// TwinCAT 3 PLC project Robotino_PLC
// ProgramVersion: 3.1.4022.0
// libraries:
//   Tc2_EtherCAT, * (Beckhoff Automation GmbH)
//   Tc2_SerialCom, * (Beckhoff Automation GmbH)
//   Tc2_Standard, * (Beckhoff Automation GmbH)
//   Tc2_System, * (Beckhoff Automation GmbH)
//   Tc2_Utilities, * (Beckhoff Automation GmbH)
//   Tc3_Module, * (Beckhoff Automation GmbH)
// project tree:
//   DUTs/ EnumState.TcDUT
//   / PlcTask.TcTTO
//   POUs/COE_Auswertung/ PDODatenMotor.TcPOU, SDODatenMotor.TcPOU, getSDODatenMotor.TcPOU, getSDOMotorErrorFlags.TcPOU, getSDODatenMotorklemme.TcPOU, SDOMotorErrorFlags.TcPOU
//   POUs/Greiferansteuerung/ Greiferansteuerung.TcPOU
//   POUs/Motoransteuerung/ Motoransteuerung.TcPOU
//   POUs/Motormesswerte/ Motormesswerte.TcPOU
//   POUs/RS232/ BackgroundPcCOM.TcPOU, FB_SerialCom.TcPOU, RS232_Communication.TcPOU
//   POUs/Shutdown/ Shutdown.TcPOU
//   POUs/UDP/ UDP.TcPOU, UDPConnect.TcPOU
// real-time tasks:
//   TASK IrSensorTask: cycle T#1ms, priority 2, ADS port 351
//   TASK UdpTask: cycle T#2ms, priority 3, ADS port 355
//   TASK SimulinkTask: cycle T#5ms, priority 4, ADS port 353
//   TASK PlcTask1: cycle T#400us, priority 1, ADS port 352
// I/O:
//   DEVICE Robotino SPS, AmsNetId 192.168.0.109.2.1
//     Klemme 1 (EK1200) [EK1200-5000 EtherCAT Netzteil (2A E-Bus)]
//       Motorklemme 1 [EL7342 2K. DC-Motor-Endstufe (50V, 3.5A)]
//       Motorklemme 2 [EL7342 2K. DC-Motor-Endstufe (50V, 3.5A)]
//       Digitale Eingänge [EL1008 8K. Dig. Eingang 24V, 3ms]
//       Digitale Ausgänge [EL2004 4K. Dig. Ausgang 24V, 0.5A]
//       Analoge Eingänge (8) [EL3068 8K. Ana. Eingang 0-10V]
//       Analog Eingänge (4) [EL3064 4K.Ana. Eingang 0-10V]
//       Netzklemme (5V) [EL9505 Netzteilklemme 5V]
//       Busendklemme [EL9011 Endklemme]
//   DEVICE UDP Adapter
//   DEVICE RS232
// variable links:
//   Robotino SPS <-> TcCOM Objects/Object2 (Gewerk3_Simulink_Regler)
//     Term 1 (EK1200)/Digitale Eingänge/Channel 2/Bumper <-> Input/processData[14]
//   Robotino SPS <-> irSensors/irSensors_Obj
//     Term 1 (EK1200)/Analog Eingänge (4)/AI Standard Channel 1/IR9 <-> Inputs/irInputData[8]
//     Term 1 (EK1200)/Analoge Eingänge (8)/AI Standard Channel {1..8}/IR{1..8} <-> Inputs/irInputData[{0..7}]  (8 links)
//   Robotino_PLC/Robotino_PLC Instance <-> RS232
//     PlcTask Inputs/BackgroundPcCOM.stIn_PcCom/D[{0..63}] <-> Inputs/Data{1..64}  (64 links)
//     PlcTask Inputs/BackgroundPcCOM.stIn_PcCom/SerStatus <-> Inputs/Status
//     PlcTask Outputs/BackgroundPcCOM.stOut_PcCom/D[{0..63}] <-> Outputs/Data{1..64}  (64 links)
//     PlcTask Outputs/BackgroundPcCOM.stOut_PcCom/SerCtrl <-> Outputs/Ctrl
//   Robotino_PLC/Robotino_PLC Instance <-> Robotino SPS/Term 1 (EK1200)/Analog Eingänge (4)
//     PlcTask Inputs/Shutdown.cell1 <-> AI Standard Channel 2/Zelle1
//     PlcTask Inputs/Shutdown.cell12 <-> AI Standard Channel 3/Zelle12
//   Robotino_PLC/Robotino_PLC Instance <-> Robotino SPS/Term 1 (EK1200)/Digitale Eingänge
//     PlcTask Inputs/Greiferansteuerung.greiferLichtschrankeFromIO <-> Channel 6/Lichtschranke
//     PlcTask Inputs/Greiferansteuerung.greiferSliderFromIO <-> Channel 5/Greifer
//     PlcTask Inputs/Motoransteuerung.bumper <-> Channel 2/Bumper
//     PlcTask Inputs/Shutdown.shutdownButton <-> Channel 8/Shutdown
//   Robotino_PLC/Robotino_PLC Instance <-> Robotino SPS/Term 1 (EK1200)/Motorklemme 1
//     PlcTask Inputs/Motormesswerte.encDataFromMotor1 <-> ENC Status compact Channel 1/Counter value
//     PlcTask Inputs/Motormesswerte.encDataFromMotor2 <-> ENC Status compact Channel 2/Counter value
//     PlcTask Inputs/PDODatenMotor.SpannungPDOMotor1 <-> DCM Synchron info data Channel 1/SpannungM1
//     PlcTask Inputs/PDODatenMotor.SpannungPDOMotor2 <-> DCM Synchron info data Channel 2/SpannungM2
//     PlcTask Inputs/PDODatenMotor.StromPDOMotor1 <-> DCM Synchron info data Channel 1/StromM1
//     PlcTask Outputs/Motoransteuerung.enableToMotor1 <-> DCM Control Channel 1/Control/Enable
//     PlcTask Outputs/Motoransteuerung.enableToMotor2 <-> DCM Control Channel 2/Control/Enable
//     PlcTask Outputs/Motoransteuerung.velocityToMotor1 <-> DCM Velocity Channel 1/Velocity
//     PlcTask Outputs/Motoransteuerung.velocityToMotor2 <-> DCM Velocity Channel 2/Velocity
//   Robotino_PLC/Robotino_PLC Instance <-> Robotino SPS/Term 1 (EK1200)/Motorklemme 2
//     PlcTask Inputs/Motormesswerte.encDataFromMotor3 <-> ENC Status compact Channel 1/Counter value
//     PlcTask Inputs/PDODatenMotor.SpannungPDOGreifer <-> DCM Synchron info data Channel 2/SpannungGreifer
//     PlcTask Inputs/PDODatenMotor.SpannungPDOMotor3 <-> DCM Synchron info data Channel 1/SpannungM3
//     PlcTask Inputs/PDODatenMotor.StromPDOGreifer <-> DCM Synchron info data Channel 2/StromGreifer
//     PlcTask Outputs/Greiferansteuerung.greiferEnable <-> DCM Control Channel 2/Control/Enable
//     PlcTask Outputs/Greiferansteuerung.greiferValue <-> DCM Velocity Channel 2/Velocity
//     PlcTask Outputs/Motoransteuerung.enableToMotor3 <-> DCM Control Channel 1/Control/Enable
//     PlcTask Outputs/Motoransteuerung.velocityToMotor3 <-> DCM Velocity Channel 1/Velocity
//   Robotino_PLC/Robotino_PLC Instance <-> TcCOM Objects/Object2 (Gewerk3_Simulink_Regler)
//     PlcTask Inputs/Greiferansteuerung.greiferSignal <-> Output/Grabber
//     PlcTask Inputs/Motoransteuerung.vThetaCartesianToMotors <-> Output/vThetaToMotors
//     PlcTask Inputs/Motoransteuerung.vXCartesianToMotors <-> Output/vXToMotors
//     PlcTask Inputs/Motoransteuerung.vYCartesianToMotors <-> Output/vYToMotors
//     PlcTask Outputs/Greiferansteuerung.greiferLichtschrankeToSimulink <-> Input/processData[0]
//     PlcTask Outputs/Greiferansteuerung.greiferSliderToSimulink <-> Input/processData[1]
//     PlcTask Outputs/Motormesswerte.vXCartesianFromMotors <-> Input/processData[2]
//     PlcTask Outputs/Motormesswerte.vYCartesianFromMotors <-> Input/processData[3]
//     PlcTask Outputs/Motormesswerte.vthetaCartesianFromMotors <-> Input/processData[4]
//     PlcTask Outputs/UDP.theta[4] <-> Input/UDP[11]
//     PlcTask Outputs/UDP.x[4] <-> Input/UDP[9]
//     PlcTask Outputs/UDP.y[4] <-> Input/UDP[10]
//   TcCOM Objects/Object2 (Gewerk3_Simulink_Regler) <-> irSensors/irSensors_Obj
//     Input/processData[{5..13}] <-> Outputs/irDistance[{0..8}]  (9 links)

CONFIGURATION Robotino_PLC
    RESOURCE PLC ON TwinCAT3
        TASK PlcTask(INTERVAL := T#400us, PRIORITY := 1);
        PROGRAM SDODatenMotor WITH PlcTask : SDODatenMotor;
        PROGRAM Motormesswerte WITH PlcTask : Motormesswerte;
        PROGRAM UDP WITH PlcTask : UDP;
        PROGRAM Greiferansteuerung WITH PlcTask : Greiferansteuerung;
        PROGRAM Motoransteuerung WITH PlcTask : Motoransteuerung;
        PROGRAM Shutdown WITH PlcTask : Shutdown;
        PROGRAM PDODatenMotor WITH PlcTask : PDODatenMotor;
        PROGRAM RS232_Communication WITH PlcTask : RS232_Communication;
    END_RESOURCE
END_CONFIGURATION

// ---- DUTs/EnumState.TcDUT
{attribute 'qualified_only'}
{attribute 'strict'}
TYPE EnumState :
(
	init,
	drive,
	reset
);
END_TYPE

// ---- POUs/COE_Auswertung/SDODatenMotor.TcPOU
PROGRAM SDODatenMotor
VAR
	DatenMotor1: getSDODatenMotor;
	DatenMotor2: getSDODatenMotor;
	DatenMotor3: getSDODatenMotor;
	
	StromMotor1 AT%Q* : INT;
	StromMotor2 AT%Q* : INT;
	StromMotor3 AT%Q* : INT;
	
	SpannungMotor1 AT%Q*:UINT;
	SpannungMotor2 AT%Q*:UINT;
	SpannungMotor3 AT%Q*:UINT;
	
END_VAR

(*** Daten azyklisch aus Klemme auslesen per SDO
	getSDO* liest CoE-Daten aus der Klemme aus:
		- getSDODatenMotor: Alle Daten, die in Objekt 9020 bzw. 9030 der Motorklemme liegen (siehe Reiter CoE-Daten auf Klemme)
			- Strom/Spannung werden alle 0.4 ms ausgelesen, Rest alle 1 ms
		- getSDODatenMotorklemme: evtl. interessante Klemmendaten, Abruf alle 5 ms
		- getSDOMotorErrorFlags: Fehlerflags wie Kurzschluss, zu hohe Temp, Überlast usw., Abruf alle 5 ms
*)

DatenMotor1.nSlaveAddr := 1001;		// Klemme  1
DatenMotor1.nIndex := 16#9020;		// Channel 1
DatenMotor1();


DatenMotor2.nSlaveAddr := 1001;		// Klemme  1
DatenMotor2.nIndex := 16#9030;		// Channel 2
DatenMotor2();

DatenMotor3.nSlaveAddr := 1002; 	// Klemme  2
DatenMotor3.nIndex := 16#9020;		// Channel 1
DatenMotor3();


StromMotor1 := DatenMotor1.Strom;
StromMotor2 := DatenMotor2.Strom;
StromMotor3 := DatenMotor3.Strom;

SpannungMotor1 :=DatenMotor1.Spannung;
SpannungMotor2 :=DatenMotor2.Spannung;
SpannungMotor3 :=DatenMotor3.Spannung;

END_PROGRAM

// ---- POUs/COE_Auswertung/getSDODatenMotor.TcPOU
FUNCTION_BLOCK getSDODatenMotor
VAR_INPUT
	nSlaveAddr: UINT;
	nIndex: WORD;
END_VAR

VAR_OUTPUT
	// Ausglesene SDOs aus 9020 bzw. 9030
	Spannung: UINT;
	Strom: INT;
	Strombegrenzung: UINT;
	Regelfehler: INT;
	Geschwindigkeit: INT;
	Overloadtime: UINT;
	Overtemperature: BOOL;
	Torqueoverload: BOOL;
	Shortcircuit: BOOL;
END_VAR
	
VAR
	MotorspannungBlock: FB_EcCoESdoRead;	
	MotorstromBlock: FB_EcCoESdoRead;
	StrombegrenzungBlock: FB_EcCoESdoRead;
	RegelfehlerBlock: FB_EcCoESdoRead;
	GeschwindigkeitBlock: FB_EcCoESdoRead;
	OverloadTimeBlock: FB_EcCoESdoRead;
	Short_CircuitBlock: FB_EcCoESdoRead;
	Torque_OverloadBlock: FB_EcCoESdoRead;
	Over_TemperatureBlock: FB_EcCoESdoRead;

	trigger: BOOL;
	triggerStromSpannung: BOOL;
	TON_0: TON;
	TON_1: TON;
	TON_2: TON;
	TON_3: TON;
	ms: TIME;

END_VAR

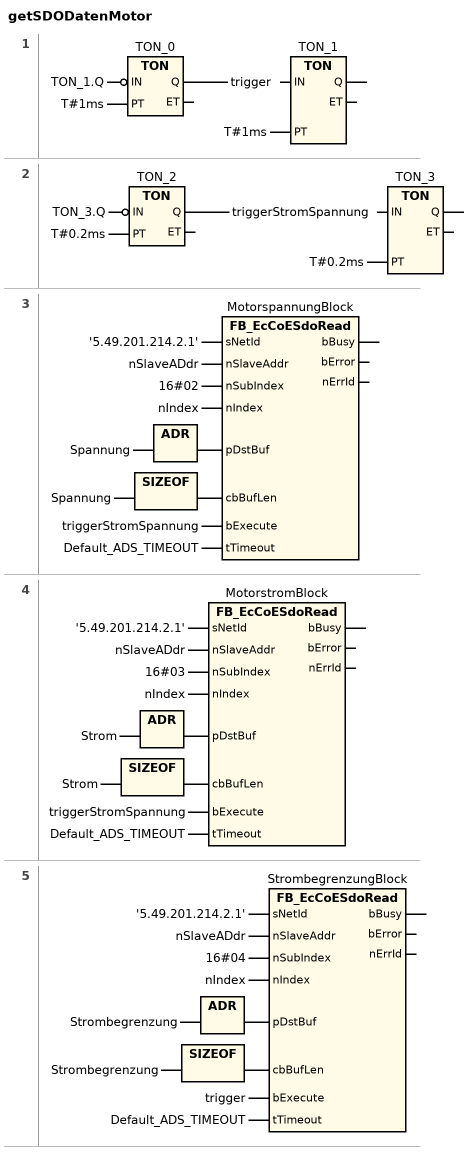
// NETWORK 1
TON_0(IN := NOT TON_1.Q, PT := T#1ms); // TON
trigger := TON_0.Q;
TON_1(IN := TON_0.Q, PT := T#1ms); // TON

// NETWORK 2
TON_2(IN := NOT TON_3.Q, PT := T#0.2ms); // TON
triggerStromSpannung := TON_2.Q;
TON_3(IN := TON_2.Q, PT := T#0.2ms); // TON

// NETWORK 3
MotorspannungBlock(
    sNetId := '5.49.201.214.2.1',
    nSlaveAddr := nSlaveADdr,
    nSubIndex := 16#02,
    nIndex := nIndex,
    pDstBuf := ADR(Spannung),
    cbBufLen := SIZEOF(Spannung),
    bExecute := triggerStromSpannung,
    tTimeout := Default_ADS_TIMEOUT); // FB_EcCoESdoRead

// NETWORK 4
MotorstromBlock(
    sNetId := '5.49.201.214.2.1',
    nSlaveAddr := nSlaveADdr,
    nSubIndex := 16#03,
    nIndex := nIndex,
    pDstBuf := ADR(Strom),
    cbBufLen := SIZEOF(Strom),
    bExecute := triggerStromSpannung,
    tTimeout := Default_ADS_TIMEOUT); // FB_EcCoESdoRead

// NETWORK 5
StrombegrenzungBlock(
    sNetId := '5.49.201.214.2.1',
    nSlaveAddr := nSlaveADdr,
    nSubIndex := 16#04,
    nIndex := nIndex,
    pDstBuf := ADR(Strombegrenzung),
    cbBufLen := SIZEOF(Strombegrenzung),
    bExecute := trigger,
    tTimeout := Default_ADS_TIMEOUT); // FB_EcCoESdoRead

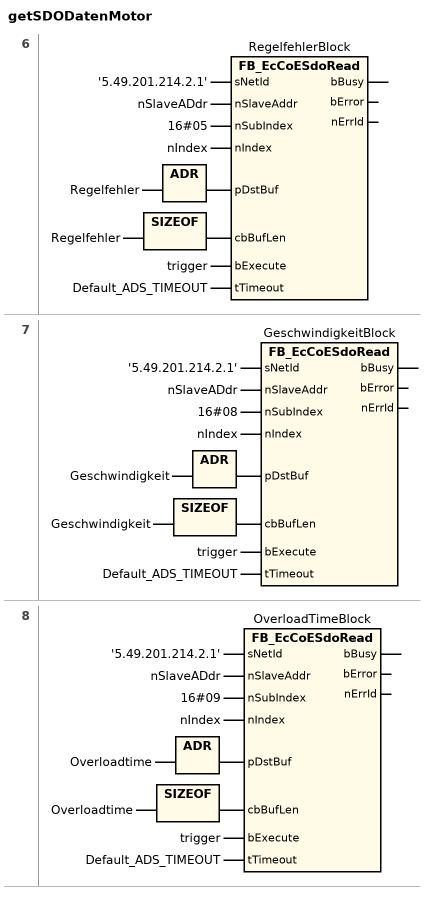
// NETWORK 6
RegelfehlerBlock(
    sNetId := '5.49.201.214.2.1',
    nSlaveAddr := nSlaveADdr,
    nSubIndex := 16#05,
    nIndex := nIndex,
    pDstBuf := ADR(Regelfehler),
    cbBufLen := SIZEOF(Regelfehler),
    bExecute := trigger,
    tTimeout := Default_ADS_TIMEOUT); // FB_EcCoESdoRead

// NETWORK 7
GeschwindigkeitBlock(
    sNetId := '5.49.201.214.2.1',
    nSlaveAddr := nSlaveADdr,
    nSubIndex := 16#08,
    nIndex := nIndex,
    pDstBuf := ADR(Geschwindigkeit),
    cbBufLen := SIZEOF(Geschwindigkeit),
    bExecute := trigger,
    tTimeout := Default_ADS_TIMEOUT); // FB_EcCoESdoRead

// NETWORK 8
OverloadTimeBlock(
    sNetId := '5.49.201.214.2.1',
    nSlaveAddr := nSlaveADdr,
    nSubIndex := 16#09,
    nIndex := nIndex,
    pDstBuf := ADR(Overloadtime),
    cbBufLen := SIZEOF(Overloadtime),
    bExecute := trigger,
    tTimeout := Default_ADS_TIMEOUT); // FB_EcCoESdoRead

END_FUNCTION_BLOCK

// ---- POUs/Motormesswerte/Motormesswerte.TcPOU
PROGRAM Motormesswerte
VAR
bStart: BOOL := FALSE;	
zaehler : UINT := 0;

//ENC Daten Differenzieren für Geschwindigkeit
diffConst:LREAL:=0.0004;//SECONDS
encDataOldMotor1:UINT:=0;
encDataOldMotor2:UINT:=0;
encDataOldMotor3:UINT:=0;

//Koordinatentransformation Weg
skalEnc:LREAL:=0.00766990393;
x1:LREAL:=0;
x2:LREAL:=0;
x3:LREAL:=0;

xFromMotor1:LREAL:=0;
xFromMotor2:LREAL:=0;
xFromMotor3:LREAL:=0;

//Koordinatentransformation Geschwindigkeit
v1:LREAL:=0;
v2:LREAL:=0;
v3:LREAL:=0;
velocityFromMotor1:LREAL:=0;
velocityFromMotor2:LREAL:=0;
velocityFromMotor3:LREAL:=0;

//INPUTS
encDataFromMotor1 AT%I*  :UINT:=0;
encDataFromMotor2 AT%I*  :UINT:=0;
encDataFromMotor3 AT%I*  :UINT:=0;

diff:  INT :=0;
diff1: INT := 0;
diff2: INT := 0;
diff3: INT := 0;

//OUTPUTS
posXCartesianFromMotors AT%Q*:LREAL:=0;
posYCartesianFromMotors AT%Q*:LREAL:=0;
posThetaCartesianFromMotors AT%Q*:LREAL:=0;

vXCartesianFromMotors AT%Q*:LREAL:=0;
vYCartesianFromMotors AT%Q*:LREAL:=0;
vthetaCartesianFromMotors AT%Q*:LREAL:=0;
END_VAR

IF bStart = FALSE THEN
	encDataOldMotor1 := encDataFromMotor1;
	encDataOldMotor2 := encDataFromMotor2;
	encDataOldMotor3 := encDataFromMotor3;
	bStart := TRUE;
END_IF



// Encoder Wegberechnung und Differenzierung für Geschwindigkeit
diff1:=UINT_TO_INT(encDataFromMotor1) - UINT_TO_INT(encDataOldMotor1);
IF diff1 >= 32767 OR diff1 <= -32767 THEN
	diff1 := 0;
	zaehler := zaehler + 1;
END_IF
diff2:=UINT_TO_INT(encDataFromMotor2) - UINT_TO_INT(encDataOldMotor2);
IF diff2 >= 32767 OR diff2 <= -32767 THEN
	diff2 := 0;
END_IF
diff3:=UINT_TO_INT(encDataFromMotor3) - UINT_TO_INT(encDataOldMotor3);
IF diff3 >= 32767 OR diff3 <= -32767 THEN
	diff3 := 0;
END_IF

xFromMotor1:=xFromMotor1+diff1*skalEnc;
velocityFromMotor1:=diff1/diffConst*skalEnc;

xFromMotor2:=xFromMotor2+diff2*skalEnc;
velocityFromMotor2:=diff2/diffConst*skalEnc;

xFromMotor3:=xFromMotor3+diff3*skalEnc;
velocityFromMotor3:=diff3/diffConst*skalEnc;

// Koordinatentransformation Weg
x1:=-xFromMotor1;
x2:=-xFromMotor2;
x3:=-xFromMotor3;

posXCartesianFromMotors:=(x3 - x1) / (2.0 * COS(30.0*PI/180));  //in mm / s
posYCartesianFromMotors:=(x1 - 2.0 * x2 + x3) / 3.0;            //in mm / s
posThetaCartesianFromMotors:=(x1 + x2 + x3) / (3.0 * 135.0);    //in rad / s

// Koordinatentransformation Geschwindigkeit
v1:=-velocityFromMotor1;
v2:=-velocityFromMotor2;
v3:=-velocityFromMotor3;

vXCartesianFromMotors:=(v3 - v1) / (2.0 * COS(30.0*PI/180));  //in mm / s
vYCartesianFromMotors:=(v1 - 2.0 * v2 + v3) / 3.0;            //in mm / s
vThetaCartesianFromMotors:=(v1 + v2 + v3) / (3.0 * 135.0);    //in rad / s

// Alte Encoderdaten speichern

encDataOldMotor1:=encDataFromMotor1;
encDataOldMotor2:=encDataFromMotor2;
encDataOldMotor3:=encDataFromMotor3;

END_PROGRAM

// ---- POUs/UDP/UDP.TcPOU
PROGRAM UDP

VAR_INPUT
	x	  AT%Q*	: ARRAY[1..4] OF LREAL;
	y	  AT%Q*	: ARRAY[1..4] OF LREAL;
	theta AT%Q*	: ARRAY[1..4] OF LREAL;
END_VAR

VAR
	udp1 : UDPConnect;
	count :INT :=0;
END_VAR

(*** UDP Kommunikation ***
	Hier wird nur der FB UDPConnect instanziert
	Für x,y,theta reichen eigentlich 8 Byte Variablen. Hier: LREAL wegen Kompatibilität
		zu Simulink Regler, der double (=LREAL) als Input braucht
*)

udp1();

END_PROGRAM

// ---- POUs/UDP/UDPConnect.TcPOU
{attribute 'c++_compatible'}
FUNCTION_BLOCK UDPConnect IMPLEMENTS ITcIoUdpProtocolRecv
VAR_INPUT
END_VAR
VAR_OUTPUT
END_VAR

VAR
	{attribute 'TcInitSymbol'}
    oid:              OTCID; 
    ipUdp:            ITcIoUdpProtocol;
    updPort:          UINT := 25000;
    nReceivedPakets:  UINT;
    hrInit :          HRESULT;
    hrSend :          HRESULT;
	
	
END_VAR

// CheckReceived() ruft ReceiveData auf

IF ipUdp <> 0 THEN
    ipUdp.CheckReceived();
END_IF

METHOD FB_exit : BOOL
VAR_INPUT
	bInCopyCode : BOOL; // if TRUE, the exit method is called for exiting an instance that is copied afterwards (online change).
END_VAR
// Destruktor für UDPConnect

IF (NOT bInCopyCode AND ipUdp <> 0) THEN //Shutdown
     ipUdp.UnregisterReceiver(updPort);
    FW_SafeRelease(ADR(ipUdp));
     FB_exit := TRUE;
ELSE
     FB_exit := FALSE;
END_IF
END_METHOD

METHOD FB_init : BOOL
VAR_INPUT
	bInitRetains : BOOL; // if TRUE, the retain variables are initialized (warm start / cold start)
	bInCopyCode : BOOL;  // if TRUE, the instance afterwards gets moved into the copy code (online change)
END_VAR

VAR
    ipSrv: ITComObjectServer;
    hr : HRESULT;
END_VAR
// Konstruktor für UDPConnect

IF NOT bInCopyCode THEN // no online change
    IF ipUdp = 0 THEN
     hrInit := FW_ObjMgr_GetObjectInstance(   oid:=oid, 
    
    iid:=TC_GLOBAL_IID_LIST.IID_ITcIoUdpProtocol, 

    pipUnk:=ADR(ipUdp) );
        IF ( SUCCEEDED(hr) AND ipUdp.RegisterReceiver(updPort, THIS^) = 0 ) THEN //open port
            FB_init := TRUE;
        ELSE
            FB_init := FALSE; 
            FW_SafeRelease(ADR(ipUdp));
        END_IF
    END_IF
END_IF
END_METHOD

METHOD FB_reinit : BOOL
VAR_INPUT
END_VAR
IF (ipUdp <> 0) THEN 
 ipUdp.RegisterReceiver(updPort, THIS^);
END_IF
END_METHOD

{attribute 'object_name' := 'ReceiveData'}
{attribute 'c++_compatible'}
{attribute 'signature_flag' := '33554688'}
{attribute 'pack_mode' := '4'}
{attribute 'show'}
{attribute 'minimal_input_size' := '4'}
METHOD ReceiveData : HRESULT
VAR_INPUT
	ipAddr	: UDINT;
	udpDestPort	: UINT;
	udpSrcPort	: UINT;
	nData	: UDINT;
	pData	: PVOID;	// Pointer auf Datenbereich des UDP-Pakets
	pVlan	: POINTER TO ETYPE_VLAN_HEADER := 0;
END_VAR

VAR
	i	: ULINT := 0;
END_VAR
nReceivedPakets := nReceivedPakets+1; 	// zählt Pakete

(*** Auslesen des Datenbereichs von UDP-Paketen ***
	* UDP-Telegramm besteht aus 56*8 = 448 Bytes (siehe UDP-Doku Lokalisierungsrechner)
	  Pro Robotino: 3*8 = 24 Bytes: je 8 Bytes für x-Koord, y-Koord, theta in rad
	  Robotino1: Bytes 1-8   -> x-Koord, Bytes 9-16  -> y-Koord, Bytes 17-24 -> theta
	  Robotino2: Bytes 25-32 -> x-Koord, Bytes 33-40 -> y-Koord, Bytes 41-48 -> theta  usw.. 
	* pData zeigt auf Adressbereich, in dem die 448 Byte großen UDP-Daten liegen
	  in der Schleife werden jeweils 8 Byte in den UDP-Array geschrieben und der Pointer nach
	  jedem Schritt um 8 Byte weiter geschoben
*)

// 4 Schleifendurchgänge für 4 Robotinos, i=0 -> Robo1 i=1 -> Robo2 usw..
FOR i := 0 TO 3 DO
	memcpy(ADR(UDP.x[i+1]),pData+((i*3)*8),8);			// x-Koord
	memcpy(ADR(UDP.y[i+1]),pData+((i*3+1)*8),8);		// y-Koord
	memcpy(ADR(UDP.theta[i+1]),pData+((i*3+2)*8),8);	// theta
END_FOR;
END_METHOD

{attribute 'c++_compatible'}
{attribute 'minimal_input_size' := '4'}
{attribute 'pack_mode' := '4'}
{warning 'Methodenimplementierung hinzufügen'}
METHOD TcAddRef : UDINT
END_METHOD

{attribute 'c++_compatible'}
{attribute 'minimal_input_size' := '4'}
{attribute 'pack_mode' := '4'}
{warning 'Methodenimplementierung hinzufügen'}
METHOD TcQueryInterface : HRESULT
VAR_INPUT
	iid	: REFERENCE TO IID;
	pipItf	: POINTER TO PVOID;
END_VAR
END_METHOD

{attribute 'c++_compatible'}
{attribute 'minimal_input_size' := '4'}
{attribute 'pack_mode' := '4'}
{warning 'Methodenimplementierung hinzufügen'}
METHOD TcRelease : UDINT
END_METHOD

END_FUNCTION_BLOCK

// ---- POUs/Greiferansteuerung/Greiferansteuerung.TcPOU
PROGRAM Greiferansteuerung
VAR
	greiferSignal AT%I*:LREAL:=0;
	greiferEnable AT%Q*:BOOL:=0;
	greiferValue  AT%Q* :INT:=0;
	
	greiferSliderFromIO 	AT%I*:BOOL:=0;
	greiferSliderToSimulink AT%Q*:LREAL:=0;
	
	greiferLichtschrankeFromIO AT%I*:BOOL:=0;
	greiferLichtschrankeToSimulink AT%Q*:LREAL:=0;
END_VAR

IF greiferSignal=0 THEN
	greiferEnable:=1;
	greiferValue:=-32767;
ELSE
	greiferEnable:=1;
	greiferValue:=32767;
END_IF

greiferSliderToSimulink:=BOOL_TO_LREAL(NOT(greiferSliderFromIO));
greiferLichtschrankeToSimulink:=BOOL_TO_LREAL(NOT(greiferLichtschrankeFromIO));

END_PROGRAM

// ---- POUs/Motoransteuerung/Motoransteuerung.TcPOU
PROGRAM Motoransteuerung
VAR	
	//Zustandsautomat
	state:		EnumState:=EnumState.init;
	nextState:	EnumState:=EnumState.init;

	//Achsen Freischalten
	
	enableMotors: BOOL	:=0;

	//Umgerechnete Werte
	vX:		LREAL:=0;
	vY:		LREAL:=0;
	vTheta:	LREAL:=0;

	//Fahrrichtung Motor
	velocityMotor1 :LREAL:=0;
	velocityMotor2 :LREAL:=0;
	velocityMotor3 :LREAL:=0;
	
	//Skalierung auf MaxGeschwindigkeit Skalierung hängt mit CoE Register 8020:07 8020:08 zusammen !!!
	velocityMax:LREAL:=942.4777961;// Nenndrehzahl U/min CoE Register 8020:07 8020:08 fesgelegt Faktor 16 Wegen Getriebe 1:16
	velocityMotorsTf:LREAL:=0;
	
	// Skalierung auf Ansteuersignale LREAL=>WORD   Skalierung hängt mit CoE Register 8020:07 8020:08 zusammen !!!
	skalPos:LREAL:=34.7668668;//  MaxValue/MaxVelocity   [1/ mm/s]   32767/(942mm/s)   MaxVelocity=D*PI*n/(16*60) //16:1 Getriebeübersetzung  
	skalNeg:LREAL:=34.76792783;//  MaxVelau/MaxVelocity   [1/ mm/s]   32768/(942mm/s)   MaxVelocity=(80mm*PI*3600 U/min)/(16*60sec/min)
	
	//Inputs: CartesianToMotors + Bumper
	vXCartesianToMotors 	AT%I*:LREAL:=0;
	vYCartesianToMotors 	AT%I*:LREAL:=0;
	vThetaCartesianToMotors AT%I*:LREAL:=0;
	bumper	   AT%I*: BOOL:=0;
	
	//Outputs: Motor Values and Enable Signal
	enableToMotor1 AT%Q*:BOOL:=FALSE;
	enableToMotor2 AT%Q*:BOOL:=FALSE;
	enableToMotor3 AT%Q*:BOOL:=FALSE;
	
	velocityToMotor1 AT%Q*:INT:=0;
	velocityToMotor3 AT%Q*:INT:=0;
	velocityToMotor2 AT%Q*:INT:=0;
	
END_VAR

(****** Konverzierung ToMotors Anfang************
Übersetzung der Koordinatentransformation aus dem Simulink Starterkit

	  conversion from positive and / or negative longitudinal, lateral and
	  rotational velocities(in milimeters per second) to three separate
	  positive motor velocities(resolution: 1Byte) and their rotation direction
inputs:  	vX  (longitudinal velocity in milimeters per second)
         	vY  (lateral velocity in milimeters per second)
			vTheta     (rotational velocity in milimeters per second)
outputs : velocityToMotor1	
			velocityToMotor2
			velocityToMotor3
conversion from longitudinal, lateral & rotational velocity to the
three separate motor velocities
*)

// Drehrichtung umgekehrt als die Richtung im alten Robotino
vX:=-vXCartesianToMotors;
vY:=-vYCartesianToMotors;
vTheta:=-vThetaCartesianToMotors;

velocityMotor1 := (-vX * COS(30.0*PI/180))	+ (vY * COS(60.0*PI/180))	+ (vTheta * 135.0);
velocityMotor2 := 0.0						+ (-vY)						+ (vTheta * 135.0);
velocityMotor3 := (vX * COS(30.0*PI/180))	+ (vY * COS(60.0*PI/180))	+ (vTheta * 135.0);

(* 	Geschwindigkeitsbegrenzung:
	Der Simulink Regler hat keine Output Begrenzung!
	Wenn Geschwindigkeit > v_max, dann muss v skaliert werden -> andere Motorgeschwindigkeiten müssen 
	dann entsprechend mitskaliert werden
	velocityMotorsTf: Faktor, der alle Geschwindigkeit auf v_max runterskaliert
*)
IF (velocityMotor1 > velocityMax) OR (velocityMotor1 < -velocityMax) THEN
    velocityMotorsTf:= velocityMotor1;
    
    velocityMotor1:= velocityMax;
    velocityMotor2:= velocityMax * velocityMotor2 / velocityMotorsTf;
    velocityMotor3:= velocityMax * velocityMotor3 / velocityMotorsTf;
END_IF

IF (velocityMotor2 > velocityMax) OR (velocityMotor2 < -velocityMax) THEN
    velocityMotorsTf:= velocityToMotor2;
    
    velocityMotor1:= velocityMax * velocityToMotor1 / velocityMotorsTf;
    velocityMotor2:= velocityMax;
    velocityMotor3:= velocityMax * velocityToMotor3 / velocityMotorsTf;
END_IF

IF (velocityMotor3 > velocityMax) OR (velocityMotor3 < -velocityMax) THEN
    velocityMotorsTf:= velocityToMotor3;
    
    velocityMotor1:= velocityMax * velocityMotor1 / velocityMotorsTf;
    velocityMotor2:= velocityMax * velocityMotor2 / velocityMotorsTf;
    velocityMotor3:= velocityMax;
END_IF
// Konvertierung ToMotors ENDE********************************************************


//MOTORANSTEUERUNG Zustandsautomat
CASE state OF
	EnumState.init:						
						IF bumper=TRUE THEN
							nextState:=EnumState.reset;
							ELSE
								nextState:=EnumState.drive;
						END_IF
	EnumState.drive:
						IF velocityMotor1>=0 THEN
							velocityToMotor1:=LREAL_TO_INT(velocityMotor1*skalPos);
						ELSE
							velocityToMotor1:=LREAL_TO_INT(velocityMotor1*skalNeg);
						END_IF
						
						IF velocityMotor2>=0 THEN
							velocityToMotor2:=LREAL_TO_INT(velocityMotor2*skalPos);
						ELSE
							velocityToMotor2:=LREAL_TO_INT(velocityMotor2*skalNeg);
						END_IF
						
						IF velocityMotor3>=0 THEN
							velocityToMotor3:=LREAL_TO_INT(velocityMotor3*skalPos);
						ELSE
							velocityToMotor3:=LREAL_TO_INT(velocityMotor3*skalNeg); 
						END_IF
							
							enableToMotor1:=1;
							enableToMotor2:=1;
							enableToMotor3:=1;
							
						IF bumper=TRUE THEN
							nextState:=EnumState.reset;
						END_IF
	EnumState.reset:
						velocityToMotor1:=0;
						velocityToMotor2:=0;
						velocityToMotor3:=0;
						enableToMotor1:=0;
						enableToMotor2:=0;
						enableToMotor3:=0;
	ELSE
		nextState:=EnumState.reset;
END_CASE
state:=nextState;

END_PROGRAM

// ---- POUs/Shutdown/Shutdown.TcPOU
PROGRAM Shutdown

VAR
	shutdownButton	AT%I* 	:BOOL := TRUE;
	cell1  			AT%I*   :INT:=0;
	cell12 			AT%I*	:INT:=0;
	
	umrechnungSpannung:LREAL:=0.000305185094; 	// 
	spannungZelle1:LREAL:=0;
	spannungZelle2:LREAL:=0;
	
	Shutdown_Block: NT_Shutdown;
END_VAR

spannungZelle1:=cell1*umrechnungSpannung;
spannungZelle2 :=(cell12-cell1)*umrechnungSpannung;

// Rudimentäre Sicherung damit Akku nicht tiefentladen wird !!!
IF(spannungZelle1<3.1 OR spannungZelle2 <3.1 OR shutdownButton = FALSE ) THEN
	Shutdown_Block(DELAY:=3,START:=TRUE);
ELSE
	Shutdown_Block(DELAY:=3,START:=FALSE);
END_IF

END_PROGRAM

// ---- POUs/COE_Auswertung/PDODatenMotor.TcPOU
PROGRAM PDODatenMotor
VAR
	StromPDOMotor1 AT%I* 		: INT;
	SpannungPDOMotor1 AT%I*		: UINT;
	StromPDOMotor2 AT%I* 		: INT;
	SpannungPDOMotor2 AT%I*	 	: UINT;
	StromPDOMotor3 AT%I* 		: INT;
	SpannungPDOMotor3 AT%I*		: UINT;
	
	StromPDOGreifer AT%I*		: INT;
	SpannungPDOGreifer AT%I*	: UINT;
END_VAR

(*	Strom und Spannung des Motors werden direkt per PDO-Mapping als Outputs gemappt
	Hier: nur Input Variablen definiert, um die Daten im Scope Server anzeigen zu lassen
*)

END_PROGRAM

// ---- POUs/RS232/RS232_Communication.TcPOU
PROGRAM RS232_Communication
VAR
	fbPcCom		: FB_SerialCom;
	
	(* exchange buffers with background communication with the PC COM port device *)
	RxBufferPcCom	: ComBuffer;	(* Receive data buffer; used with all receive function blocks *)
	TxBufferPcCom	: ComBuffer;	(* Transmit data buffer; used with all receive function blocks *)
END_VAR

(*** RS232 Kommunikationsbeispiel ***
	BackhgroundPcCOM: Hintergrundprogramm, das zyklisch mit COM-Schnittstelle des IPC kommuniziert
	fbPcCom: FB zum Senden und Empfangen von Daten
*)
BackgroundPcCOM(RxBufferPcCom:=RxBufferPcCom, TxBufferPcCom:=TxBufferPcCom);
fbPcCom(TxBuffer:=TxBufferPcCom, RxBuffer:=RxBufferPcCom);

END_PROGRAM

// ---- POUs/RS232/FB_SerialCom.TcPOU
FUNCTION_BLOCK FB_SerialCom
VAR_IN_OUT
	TxBuffer	: ComBuffer;
	RxBuffer	: ComBuffer;
END_VAR
VAR
	Timer		: TON := (PT:=T#5S); // Timer für Sendezyklus
	fbSend		: SendString;
	bSendBusy	: BOOL;
	eSendErrorID: ComError_t;

	(* 	ReceiveString kann 80 Zeichen empfangen
		Wenn mehr Platz gebraucht: -> ReceiveString255 *)
	fbReceive		: ReceiveString;
	sReceivedString	: STRING;
	sLastReceivedString: STRING;
	bStringReceived	: BOOL;
	bReceiveBusy	: BOOL;
	bReceiveError	: BOOL;
	eReceiveErrorID	: ComError_t;
	bReceiveTimeout	: BOOL;
	nReceiveCounter	: UDINT;
END_VAR

(* fbSend wird alle x Sekunden aktiviert, um den Sendstring zu senden
   fbSend wird auch aktiviert, wenn der String nach einem Zyklus noch nicht fertig gesendet wurde
   (d.h. wenn Busy = True ist)
*)
Timer(IN:=TRUE);
IF Timer.Q OR fbSend.Busy THEN
	Timer(IN:=FALSE); (* reset timer *)
	fbSend(
			SendString:= 'Hello World! Here I am! Go Robo!!!#',  // Hier Nachricht definieren
			TXbuffer:= TxBuffer,
			Busy=> bSendBusy,
			Error=> );
	IF fbSend.Error <> COMERROR_NOERROR THEN
		eSendErrorID := fbSend.Error;
	END_IF
END_IF

(* fbReceive empfängt Daten, die mit \02 anfangen und \03 aufhören
	Prefix und Suffix können auch anders gewählt werden oder leer sein
	(leer -> fbReceive empfängt dauerhaft)
*)
fbReceive(	
	Prefix:= '$02',	// $02 == \02 ascii
	Suffix:= '$03',	// $03 == \03 ascii
	Timeout:= T#3S,
	ReceivedString:= sReceivedString, // empfangene Nachricht
	RXbuffer:= RxBuffer,
	StringReceived=> bStringReceived,
	Busy=> bReceiveBusy,
	Error=> ,
	RxTimeout=> bReceiveTimeout );
IF fbReceive.Error <> COMERROR_NOERROR THEN
	eReceiveErrorID := fbReceive.Error;
END_IF

// Counter how many messages are recieved
IF bStringReceived THEN
	nReceiveCounter := nReceiveCounter + 1;
	sLastReceivedString := sReceivedString;
END_IF

END_FUNCTION_BLOCK

// ---- POUs/RS232/BackgroundPcCOM.TcPOU
PROGRAM BackgroundPcCOM
VAR_IN_OUT
	RxBufferPcCom		: ComBuffer;	(* Receive data buffer; used with all receive function blocks *)
	TxBufferPcCom		: ComBuffer;	(* Transmit data buffer; used with all receive function blocks *)
END_VAR
VAR
	(* background communication with the PC COM port device *)
	fbPcComCtrl			: SerialLineControl;
	bPcComCtrlError		: BOOL;
	ePcComCtrlErrorID	: ComError_t;	
	(* 	I/O variables for a PC-COM port *)
	stIn_PcCom AT %I*	: PcComInData;	(* linked to the port in the TwinCAT System Manager *)
	stOut_PcCom AT %Q*	: PcComOutData;	(* linked to the port in the TwinCAT System Manager *)
END_VAR

(*
The SerialLineControl function block is supposed to be called in every PLC cycle.
It communicates with the serial line hardware device and transmits or receives data.
The SerialLineControl can be called in the standard task (e.g.for PcCOM port usage) 
or in a separate fast task (e.g.for terminal usage) as well.
A fast separate task will be necessary at high baud rates or with KL6001 terminals 
which have a small process image (3 or 5 data bytes only)
*)

(* background communication with the PC COM port device *)
fbPcComCtrl(
	Mode:= SERIALLINEMODE_PC_COM_PORT, 
	pComIn:= ADR(stIn_PcCom), 
	pComOut:= ADR(stOut_PcCom), 
	SizeComIn:= SIZEOF(stIn_PcCom), 
	Error=> , 
	ErrorID=> , 
	TxBuffer:= TxBufferPcCom, 
	RxBuffer:= RxBufferPcCom );
IF fbPcComCtrl.Error THEN
	bPcComCtrlError := TRUE;
	ePcComCtrlErrorID := fbPcComCtrl.ErrorID;
END_IF

END_PROGRAM

// ---- POUs/COE_Auswertung/getSDOMotorErrorFlags.TcPOU
FUNCTION_BLOCK getSDOMotorErrorFlags
VAR_INPUT
	nSlaveAddr: UINT;
	nIndex: WORD;
END_VAR

VAR_OUTPUT
	Overtemp: BOOL;
	Torqueoverload: BOOL;
	Shortcircuit: BOOL;
	
END_VAR
VAR

	Short_CircuitBlock: FB_EcCoESdoRead;
	Torque_OverloadBlock: FB_EcCoESdoRead;
	Over_TemperatureBlock: FB_EcCoESdoRead;

	trigger: BOOL;
	TON_0: TON;
	TON_1: TON;
	ms: TIME;

END_VAR

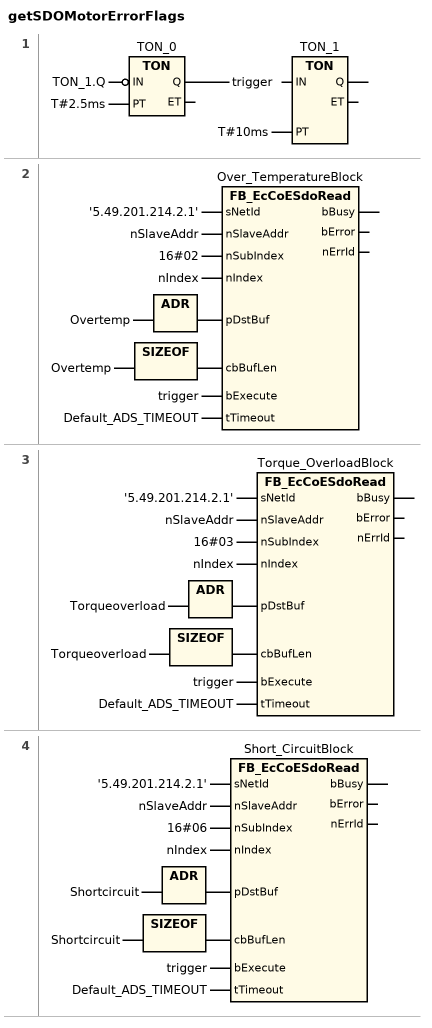
// NETWORK 1
TON_0(IN := NOT TON_1.Q, PT := T#2.5ms); // TON
trigger := TON_0.Q;
TON_1(IN := TON_0.Q, PT := T#10ms); // TON

// NETWORK 2
Over_TemperatureBlock(
    sNetId := '5.49.201.214.2.1',
    nSlaveAddr := nSlaveAddr,
    nSubIndex := 16#02,
    nIndex := nIndex,
    pDstBuf := ADR(Overtemp),
    cbBufLen := SIZEOF(Overtemp),
    bExecute := trigger,
    tTimeout := Default_ADS_TIMEOUT); // FB_EcCoESdoRead

// NETWORK 3
Torque_OverloadBlock(
    sNetId := '5.49.201.214.2.1',
    nSlaveAddr := nSlaveAddr,
    nSubIndex := 16#03,
    nIndex := nIndex,
    pDstBuf := ADR(Torqueoverload),
    cbBufLen := SIZEOF(Torqueoverload),
    bExecute := trigger,
    tTimeout := Default_ADS_TIMEOUT); // FB_EcCoESdoRead

// NETWORK 4
Short_CircuitBlock(
    sNetId := '5.49.201.214.2.1',
    nSlaveAddr := nSlaveAddr,
    nSubIndex := 16#06,
    nIndex := nIndex,
    pDstBuf := ADR(Shortcircuit),
    cbBufLen := SIZEOF(Shortcircuit),
    bExecute := trigger,
    tTimeout := Default_ADS_TIMEOUT); // FB_EcCoESdoRead

END_FUNCTION_BLOCK

// ---- POUs/COE_Auswertung/getSDODatenMotorklemme.TcPOU
FUNCTION_BLOCK getSDODatenMotorklemme
VAR_INPUT
	nSlaveAddr: UINT;
END_VAR
VAR_OUTPUT
	
	Motorklemme1Internaltemperature: SINT;
	Motorklemme1Steuerspannung: UINT;
	Motorklemme1Lastspannung: UINT;
	Motorklemme1Zykluszeit: UINT;
	Motorklemme1PWMFrequency: UINT;
		
END_VAR
VAR

	Internal_Temperature: FB_EcCoESdoRead;
	Control_Voltage: FB_EcCoESdoRead;
	Supply_Voltage: FB_EcCoESdoRead;
	Cycletime: FB_EcCoESdoRead;
	PWM_Frequency: FB_EcCoESdoRead;
	
	trigger: BOOL;
	TON_0: TON;
	TON_1: TON;
	ms: TIME;

END_VAR

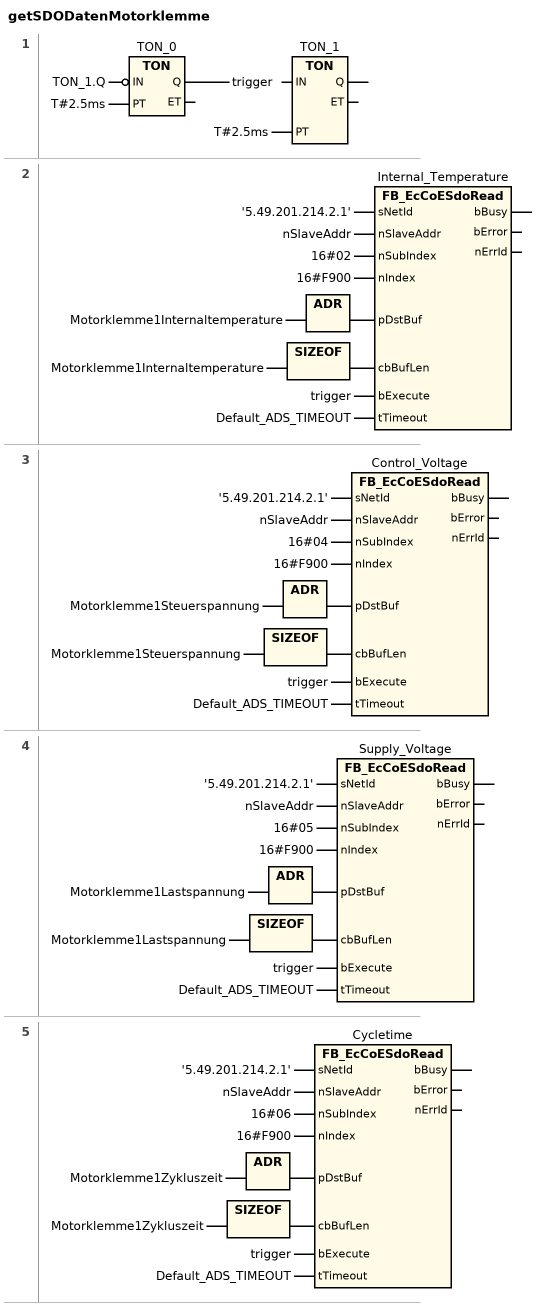
// NETWORK 1
TON_0(IN := NOT TON_1.Q, PT := T#2.5ms); // TON
trigger := TON_0.Q;
TON_1(IN := TON_0.Q, PT := T#2.5ms); // TON

// NETWORK 2
Internal_Temperature(
    sNetId := '5.49.201.214.2.1',
    nSlaveAddr := nSlaveAddr,
    nSubIndex := 16#02,
    nIndex := 16#F900,
    pDstBuf := ADR(Motorklemme1Internaltemperature),
    cbBufLen := SIZEOF(Motorklemme1Internaltemperature),
    bExecute := trigger,
    tTimeout := Default_ADS_TIMEOUT); // FB_EcCoESdoRead

// NETWORK 3
Control_Voltage(
    sNetId := '5.49.201.214.2.1',
    nSlaveAddr := nSlaveAddr,
    nSubIndex := 16#04,
    nIndex := 16#F900,
    pDstBuf := ADR(Motorklemme1Steuerspannung),
    cbBufLen := SIZEOF(Motorklemme1Steuerspannung),
    bExecute := trigger,
    tTimeout := Default_ADS_TIMEOUT); // FB_EcCoESdoRead

// NETWORK 4
Supply_Voltage(
    sNetId := '5.49.201.214.2.1',
    nSlaveAddr := nSlaveAddr,
    nSubIndex := 16#05,
    nIndex := 16#F900,
    pDstBuf := ADR(Motorklemme1Lastspannung),
    cbBufLen := SIZEOF(Motorklemme1Lastspannung),
    bExecute := trigger,
    tTimeout := Default_ADS_TIMEOUT); // FB_EcCoESdoRead

// NETWORK 5
Cycletime(
    sNetId := '5.49.201.214.2.1',
    nSlaveAddr := nSlaveAddr,
    nSubIndex := 16#06,
    nIndex := 16#F900,
    pDstBuf := ADR(Motorklemme1Zykluszeit),
    cbBufLen := SIZEOF(Motorklemme1Zykluszeit),
    bExecute := trigger,
    tTimeout := Default_ADS_TIMEOUT); // FB_EcCoESdoRead

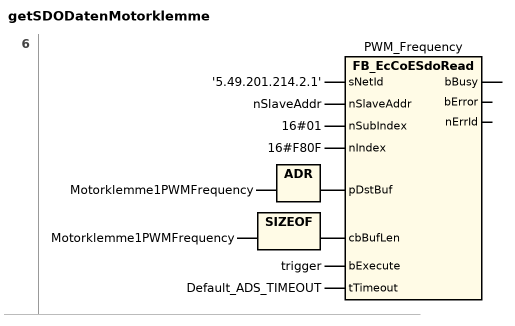
// NETWORK 6
PWM_Frequency(
    sNetId := '5.49.201.214.2.1',
    nSlaveAddr := nSlaveAddr,
    nSubIndex := 16#01,
    nIndex := 16#F80F,
    pDstBuf := ADR(Motorklemme1PWMFrequency),
    cbBufLen := SIZEOF(Motorklemme1PWMFrequency),
    bExecute := trigger,
    tTimeout := Default_ADS_TIMEOUT); // FB_EcCoESdoRead

END_FUNCTION_BLOCK

// ---- POUs/COE_Auswertung/SDOMotorErrorFlags.TcPOU
PROGRAM SDOMotorErrorFlags
VAR
	ErrorFlagsKlemme1: getSDOMotorErrorFlags;
	ErrorFlagsKlemme2: getSDOMotorErrorFlags;
END_VAR

ErrorFlagsKlemme1.nSlaveAddr := 1002;
ErrorFlagsKlemme1();

END_PROGRAM
